(* CODESYS project e!C_BasicProg_1.ECP

Project tree, tasks and I/O mapping:
  PFC8203 : 750-8203 PFC200 2ETH CAN, WAGO, order no. 0750-8203, version 5.11.1.16
    application Application
      libraries: Standard, * (System); Util, * (System)
      task Test (cyclic, interval T#10ms, priority 11) calls PLC_PRG
      task VISU_TASK (cyclic, interval 100 ms, priority 15) calls VisuElems.Visu_Prg
      Data types/
        data type typControlInterface
      Global Variables/
        global variables Variable_Configuration
        global variables GVL
      POUs/
        CASE_OF/
          program Template_CASE_OF [ST]
          program Test1_CASE_OF [ST]
        FB_POINTER/
          function block fbPointerControl [ST]
          program Template_FB_POINTER [ST]
          program Test1_FB_POINTER [ST]
        FB_STRUCT/
          function block fbStructControl [ST]
          program Template_FB_STRUCT [ST]
          program Test1_FB_STRUCT [ST]
        FOR_DO_ARRAY/
          program Template_FOR_DO_ARRAY [ST]: Action1_ST, Action2_ST, Action3_ST
          program Test1_FOR_DO_ARRAY [ST]: Action1_ST, Action2_ST, Action3_ST
        program PLC_PRG [ST]
        IF_THEN_ELSE/
          program Test1_IF_THEN_ELSE [ST]: Action3_CFC, Action1_ST, Action2_SFC, ActivationMonitoring_active, Inactivation_active, Init_active, OutputControl_active
          program Template_IF_THEN_ELSE [ST]: Action2_SFC, Action3_CFC, Action1_ST, Inactivation_active, ActivationMonitoring_active, OutputControl_active, Init_active
      Visualizations/
        visualisation FB_STRUCT
        visualisation IF_THEN_ELSE
      global variables PersistentVars
      trace Sampling_Trace (task Test): Test_FB_STRUCT.typEngineControl.rControlPosition, Test1_FOR_DO_ARRAY.rSineSample
    DeviceAdapter
    Kbus : Kbus, WAGO, version 1.4.0.2
        unmapped channels: K-BUS diagnostics
    MODBUS
      MODBUS : MODBUS, WAGO, order no. n/a, version 1.1.1.15
    CANbus
  libraries: Util, 3.5.11.0 (System); VisuSymbols, 3.5.10.0 (System); WagoVisuIcons, 1.0.0.8 (WAGO)
  GlobalImagePool
  text list GlobalTextList
*)

// PFC8203/Application/Data types/typControlInterface
TYPE typControlInterface :
STRUCT
	TON_ControlDelay: TON;
	R_TRIG_ControlStart: R_TRIG;
	R_TRIG_ControlStop: R_TRIG;
	tControlDelay: TIME := T#2s;
	xControlEnable: BOOL;
	xControlRun: BOOL;
	xControlStart: BOOL;
	xControlStop: BOOL;
	xControlOut: BOOL;

	GEN_ControlSimulator: GEN;
	SimulatorMode: GEN_MODE;
	SimulatorPeriod: TIME := T#2s;
	SimulatorAmplitude: INT := 100;
	rSimulatorLimit: REAL := 100.0;
	rSimulatorLevel: REAL := 100.1;
	rSimulatorPosition: REAL;
END_STRUCT
END_TYPE

// PFC8203/Application/Global Variables/Variable_Configuration
VAR_CONFIG
END_VAR

// PFC8203/Application/PersistentVars
VAR_GLOBAL PERSISTENT RETAIN
END_VAR

// PFC8203/Application/Global Variables/GVL
VAR_GLOBAL
END_VAR

// PFC8203/Application/POUs/PLC_PRG
PROGRAM PLC_PRG
VAR
END_VAR



Template_IF_THEN_ELSE();
Test1_IF_THEN_ELSE();

Template_CASE_OF();
Test1_CASE_OF();


Template_FOR_DO_ARRAY();
Test1_FOR_DO_ARRAY();


Template_FB_STRUCT();
Test1_FB_STRUCT();


Template_FB_POINTER();
Test1_FB_POINTER();

END_PROGRAM

// PFC8203/Application/POUs/IF_THEN_ELSE/Template_IF_THEN_ELSE
PROGRAM Template_IF_THEN_ELSE
VAR
	TON_ControlDelay_1: TON;
	R_TRIG_ControlStart_1: R_TRIG;
	R_TRIG_ControlStop_1: R_TRIG;
	tControlDelay_1: TIME := T#2s;
	xControlEnable_1: BOOL;
	xControlRun_1: BOOL;
	xControlStart_1: BOOL;
	xControlStop_1: BOOL;
	xControlOut_1: BOOL;

	TON_ControlDelay_2: TON;
	R_TRIG_ControlStart_2: R_TRIG;
	R_TRIG_ControlStop_2: R_TRIG;
	tControlDelay_2: TIME := T#2s;
	xControlEnable_2: BOOL;
	xControlRun_2: BOOL;
	xControlStart_2: BOOL;
	xControlStop_2: BOOL;
	xControlOut_2: BOOL;

	TON_ControlDelay_3: TON;
	R_TRIG_ControlStart_3: R_TRIG;
	R_TRIG_ControlStop_3: R_TRIG;
	tControlDelay_3: TIME := T#2s;
	xControlEnable_3: BOOL;
	xControlRun_3: BOOL;
	xControlStart_3: BOOL;
	xControlStop_3: BOOL;
	xControlOut_3: BOOL;

END_VAR
VAR // added by the converter: edge detectors and wires of the graphical bodies
    _w1 : BOOL;
END_VAR



Action1_ST();

Action2_SFC();

Action3_CFC();

ACTION Action2_SFC:
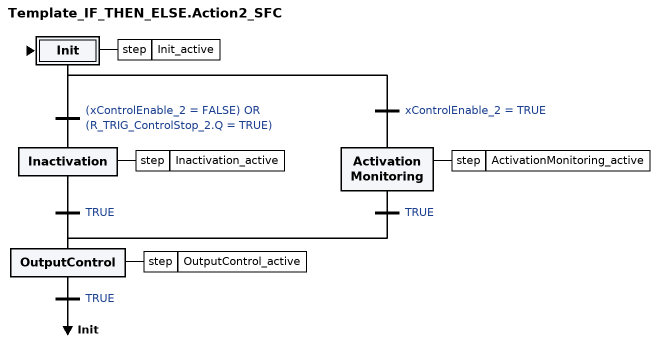
INITIAL_STEP Init:
    Init_active(N);  // step action
END_STEP
TRANSITION FROM Init TO Inactivation
    := (xControlEnable_2 = FALSE) OR (R_TRIG_ControlStop_2.Q = TRUE);
END_TRANSITION
STEP Inactivation:
    Inactivation_active(N);  // step action
END_STEP
TRANSITION FROM Inactivation TO OutputControl
    := TRUE;
END_TRANSITION
TRANSITION FROM Init TO ActivationMonitoring
    := xControlEnable_2 = TRUE;
END_TRANSITION
STEP ActivationMonitoring:
    ActivationMonitoring_active(N);  // step action
END_STEP
TRANSITION FROM ActivationMonitoring TO OutputControl
    := TRUE;
END_TRANSITION
STEP OutputControl:
    OutputControl_active(N);  // step action
END_STEP
TRANSITION FROM OutputControl TO Init
    := TRUE;
END_TRANSITION
// branch label Branch1_Action2_SFC
END_ACTION

ACTION Action3_CFC:
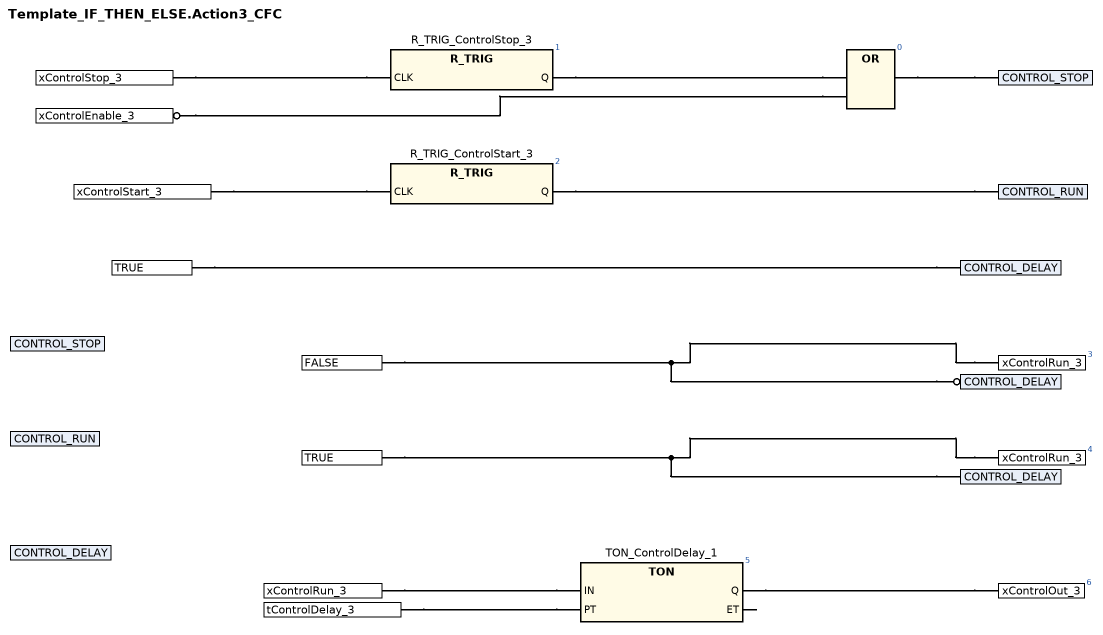
(* R_TRIG_ControlStop_3.Q OR NOT xControlEnable_3; result not used *)
R_TRIG_ControlStop_3(CLK := xControlStop_3); // R_TRIG
R_TRIG_ControlStart_3(CLK := xControlStart_3); // R_TRIG
xControlRun_3 := FALSE;
xControlRun_3 := TRUE;
TON_ControlDelay_1(IN := xControlRun_3, PT := tControlDelay_3); // TON
xControlOut_3 := TON_ControlDelay_1.Q;
END_ACTION

ACTION Action1_ST:


(* Monitor start/stop signal for output activation/inactivation *)
R_TRIG_ControlStart_1(CLK:= xControlStart_1);
R_TRIG_ControlStop_1(CLK:= xControlStop_1);
IF ((xControlEnable_1 = FALSE) OR (R_TRIG_ControlStop_1.Q = TRUE))THEN
	xControlRun_1 := FALSE;
ELSE
	IF (R_TRIG_ControlStart_1.Q = TRUE) THEN
		xControlRun_1 := TRUE;
	END_IF
END_IF


(* Activate output after specified delay *)
TON_ControlDelay_1(IN:= xControlRun_1, PT:= tControlDelay_1, Q=> xControlOut_1);
END_ACTION

ACTION Inactivation_active:
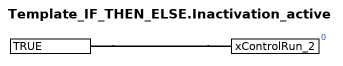
xControlRun_2 := TRUE;
END_ACTION

ACTION ActivationMonitoring_active:
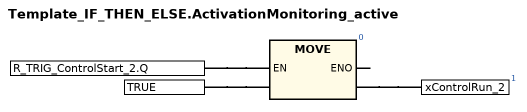
IF R_TRIG_ControlStart_2.Q THEN _w1 := TRUE; END_IF
xControlRun_2 := _w1;
END_ACTION

ACTION OutputControl_active:
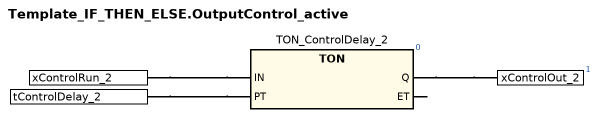
TON_ControlDelay_2(IN := xControlRun_2, PT := tControlDelay_2); // TON
xControlOut_2 := TON_ControlDelay_2.Q;
END_ACTION

ACTION Init_active:
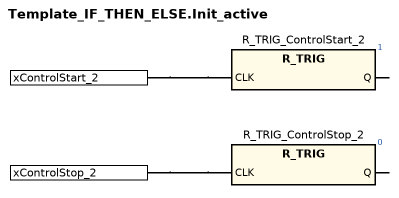
R_TRIG_ControlStop_2(CLK := xControlStop_2); // R_TRIG
R_TRIG_ControlStart_2(CLK := xControlStart_2); // R_TRIG
END_ACTION

END_PROGRAM

// PFC8203/Application/POUs/IF_THEN_ELSE/Test1_IF_THEN_ELSE
PROGRAM Test1_IF_THEN_ELSE
VAR
	TON_ControlDelay_1: TON;
	R_TRIG_ControlStart_1: R_TRIG;
	R_TRIG_ControlStop_1: R_TRIG;
	tControlDelay_1: TIME := T#2s;
	xControlEnable_1: BOOL;
	xControlRun_1: BOOL;
	xControlStart_1: BOOL;
	xControlStop_1: BOOL;
	xControlOut_1: BOOL;

	TON_ControlDelay_2: TON;
	R_TRIG_ControlStart_2: R_TRIG;
	R_TRIG_ControlStop_2: R_TRIG;
	tControlDelay_2: TIME := T#2s;
	xControlEnable_2: BOOL;
	xControlRun_2: BOOL;
	xControlStart_2: BOOL;
	xControlStop_2: BOOL;
	xControlOut_2: BOOL;

	TON_ControlDelay_3: TON;
	R_TRIG_ControlStart_3: R_TRIG;
	R_TRIG_ControlStop_3: R_TRIG;
	tControlDelay_3: TIME := T#2s;
	xControlEnable_3: BOOL;
	xControlRun_3: BOOL;
	xControlStart_3: BOOL;
	xControlStop_3: BOOL;
	xControlOut_3: BOOL;

END_VAR
VAR // added by the converter: edge detectors and wires of the graphical bodies
    _w1 : BOOL;
END_VAR



Action1_ST();

Action2_SFC();

Action3_CFC();

ACTION Action3_CFC:
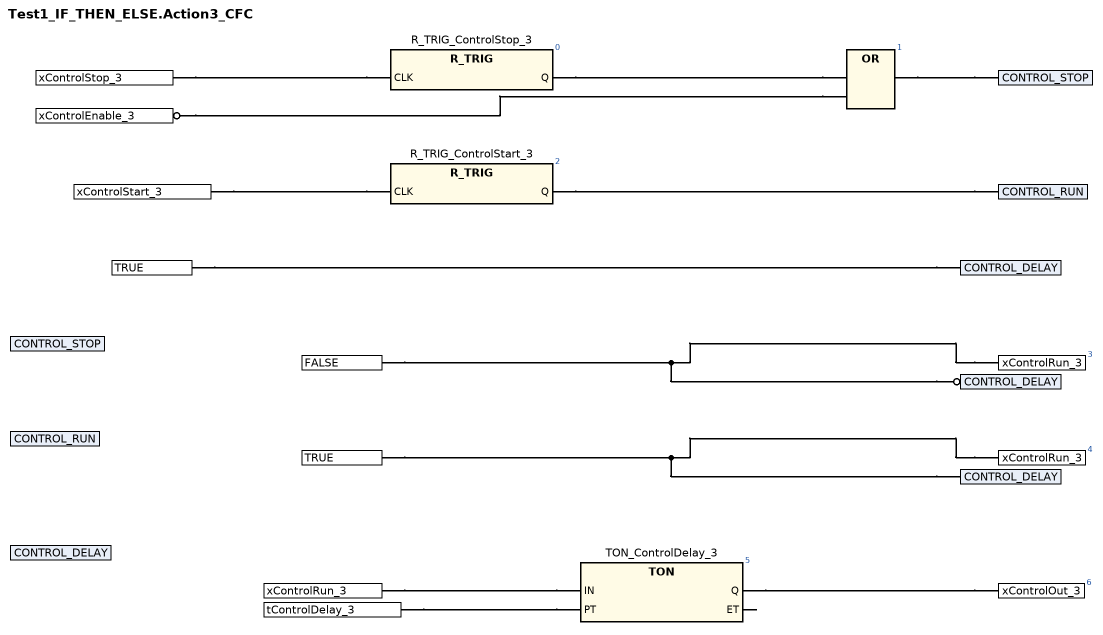
R_TRIG_ControlStop_3(CLK := xControlStop_3); // R_TRIG
(* R_TRIG_ControlStop_3.Q OR NOT xControlEnable_3; result not used *)
R_TRIG_ControlStart_3(CLK := xControlStart_3); // R_TRIG
xControlRun_3 := FALSE;
xControlRun_3 := TRUE;
TON_ControlDelay_3(IN := xControlRun_3, PT := tControlDelay_3); // TON
xControlOut_3 := TON_ControlDelay_3.Q;
END_ACTION

ACTION Action1_ST:


(* Monitor start/stop signal for output activation/inactivation *)
R_TRIG_ControlStart_1(CLK:= xControlStart_1);
R_TRIG_ControlStop_1(CLK:= xControlStop_1);
IF ((xControlEnable_1 = FALSE) OR (R_TRIG_ControlStop_1.Q = TRUE))THEN
	xControlRun_1 := FALSE;
ELSE
	IF (R_TRIG_ControlStart_1.Q = TRUE) THEN
		xControlRun_1 := TRUE;
	END_IF
END_IF


(* Activate output after specified delay *)
TON_ControlDelay_1(IN:= xControlRun_1, PT:= tControlDelay_1, Q=> xControlOut_1);
END_ACTION

ACTION Action2_SFC:
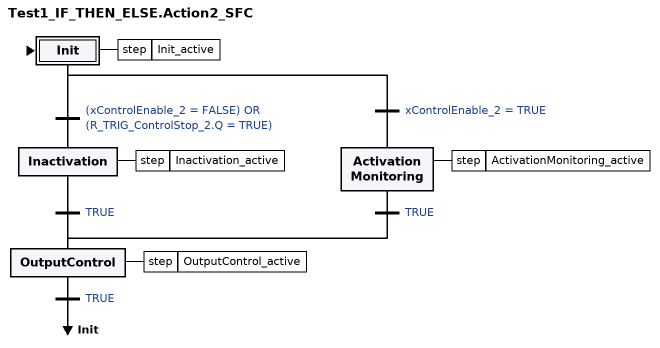
INITIAL_STEP Init:
    Init_active(N);  // step action
END_STEP
TRANSITION FROM Init TO Inactivation
    := (xControlEnable_2 = FALSE) OR (R_TRIG_ControlStop_2.Q = TRUE);
END_TRANSITION
STEP Inactivation:
    Inactivation_active(N);  // step action
END_STEP
TRANSITION FROM Inactivation TO OutputControl
    := TRUE;
END_TRANSITION
TRANSITION FROM Init TO ActivationMonitoring
    := xControlEnable_2 = TRUE;
END_TRANSITION
STEP ActivationMonitoring:
    ActivationMonitoring_active(N);  // step action
END_STEP
TRANSITION FROM ActivationMonitoring TO OutputControl
    := TRUE;
END_TRANSITION
STEP OutputControl:
    OutputControl_active(N);  // step action
END_STEP
TRANSITION FROM OutputControl TO Init
    := TRUE;
END_TRANSITION
// branch label Branch1_Action2_SFC
END_ACTION

ACTION ActivationMonitoring_active:
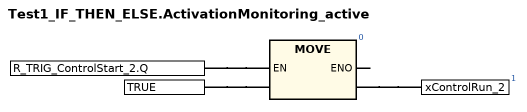
IF R_TRIG_ControlStart_2.Q THEN _w1 := TRUE; END_IF
xControlRun_2 := _w1;
END_ACTION

ACTION Inactivation_active:
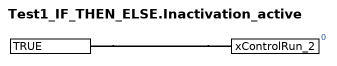
xControlRun_2 := TRUE;
END_ACTION

ACTION Init_active:
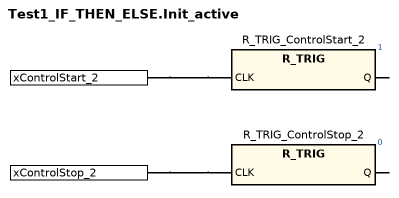
R_TRIG_ControlStop_2(CLK := xControlStop_2); // R_TRIG
R_TRIG_ControlStart_2(CLK := xControlStart_2); // R_TRIG
END_ACTION

ACTION OutputControl_active:
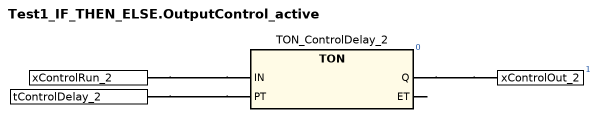
TON_ControlDelay_2(IN := xControlRun_2, PT := tControlDelay_2); // TON
xControlOut_2 := TON_ControlDelay_2.Q;
END_ACTION

END_PROGRAM

// PFC8203/Application/POUs/CASE_OF/Template_CASE_OF
PROGRAM Template_CASE_OF
VAR
	TON_ControlDelay: TON;
	R_TRIG_ControlStart: R_TRIG;
	R_TRIG_ControlStop: R_TRIG;
	tControlDelay: TIME := T#2s;
	wControlState: WORD;
	xControlEnable: BOOL;
	xControlRun: BOOL;
	xControlStart: BOOL;
	xControlStop: BOOL;
	xControlOut: BOOL;
END_VAR



R_TRIG_ControlStart(CLK:= xControlStart);
R_TRIG_ControlStop(CLK:= xControlStop);

(* Monitor signal activation sequence *)
CASE wControlState OF

	0:(* Init signal monitoring *)
		wControlState := 10;

	10:(* Signal currently active, wait for inactivation *)
		IF ((xControlEnable = FALSE) OR (R_TRIG_ControlStop.Q = TRUE)) THEN
			xControlRun := FALSE;
			wControlState := 20;
		END_IF

	20:(* Signal currently incative, wait for activation *)
		IF ((xControlEnable = TRUE) AND (R_TRIG_ControlStart.Q = TRUE)) THEN
			xControlRun := TRUE;
			wControlState := 10;
		END_IF

END_CASE


(* Activate output after specified delay when commanded *)
TON_ControlDelay(IN:= xControlRun, PT:= tControlDelay, Q=> xControlOut);

END_PROGRAM

// PFC8203/Application/POUs/CASE_OF/Test1_CASE_OF
PROGRAM Test1_CASE_OF
VAR
	TON_ControlDelay: TON;
	R_TRIG_ControlStart: R_TRIG;
	R_TRIG_ControlStop: R_TRIG;
	tControlDelay: TIME := T#2s;
	wControlState: WORD;
	xControlEnable: BOOL;
	xControlRun: BOOL;
	xControlStart: BOOL;
	xControlStop: BOOL;
	xControlOut: BOOL;
END_VAR



R_TRIG_ControlStart(CLK:= xControlStart);
R_TRIG_ControlStop(CLK:= xControlStop);

(* Monitor signal activation sequence *)
CASE wControlState OF

	0:(* Init signal monitoring *)
		wControlState := 10;

	10:(* Signal currently active, wait for inactivation *)
		IF ((xControlEnable = FALSE) OR (R_TRIG_ControlStop.Q = TRUE)) THEN
			xControlRun := FALSE;
			wControlState := 20;
		END_IF

	20:(* Signal currently incative, wait for activation *)
		IF ((xControlEnable = TRUE) AND (R_TRIG_ControlStart.Q = TRUE)) THEN
			xControlRun := TRUE;
			wControlState := 10;
		END_IF

END_CASE


(* Activate output after specified delay when commanded *)
TON_ControlDelay(IN:= xControlRun, PT:= tControlDelay, Q=> xControlOut);

END_PROGRAM

// PFC8203/Application/POUs/FOR_DO_ARRAY/Template_FOR_DO_ARRAY
PROGRAM Template_FOR_DO_ARRAY
VAR CONSTANT
	iArrayLimit1: INT := 9;
	iArrayLimit2: INT := 9;
	iArrayLimit3: INT := 19;
	iArrayLimit4: INT := 49;
	iModuloLimit: INT := 50;
END_VAR
VAR
	iArrayIndex: INT;
	dwCnt: DWORD;
	wCnt: WORD;
	awArrayTest1: ARRAY[0..iArrayLimit1] OF WORD;
	adwArrayTest2 AT %MW0 : ARRAY[0..iArrayLimit2] OF DWORD;
	awArrayTest3 AT %MW0 : ARRAY[0..iArrayLimit3] OF WORD;

	iArrayIndexModulo: INT;
	TON_SineSampler: TON;
	tSineInterval: TIME := T#200ms;
	rSineAngle: REAL;
	rSineSample: REAL;
	arSineArray: ARRAY[0..iArrayLimit4] OF REAL;

	TON_ControlDelay: ARRAY[0..iArrayLimit1] OF TON;
	R_TRIG_ControlStart: ARRAY[0..iArrayLimit1] OF R_TRIG;
	R_TRIG_ControlStop: ARRAY[0..iArrayLimit1] OF R_TRIG;
	tControlDelay: ARRAY[0..iArrayLimit1] OF TIME := [iArrayLimit1(T#2S)];
	xControlEnable: ARRAY[0..iArrayLimit1] OF BOOL;
	xControlRun: ARRAY[0..iArrayLimit1] OF BOOL;
	xControlStart: ARRAY[0..iArrayLimit1] OF BOOL;
	xControlStop: ARRAY[0..iArrayLimit1] OF BOOL;
	xControlOut: ARRAY[0..iArrayLimit1] OF BOOL;
END_VAR


Action1_ST();

Action2_ST();

Action3_ST();

ACTION Action1_ST:

(* Run same logic for all array elements *)
FOR iArrayIndex := 0 TO iArrayLimit1 DO

	wCnt := wCnt + 1;
	dwCnt := dwCnt + 1;

	awArrayTest1[iArrayIndex] := wCnt;

	adwArrayTest2[iArrayIndex] := dwCnt;

	awArrayTest3[2*iArrayIndex] := DWORD_TO_WORD(dwCnt);
	awArrayTest3[(2*iArrayIndex)+1] := DWORD_TO_WORD(SHR(dwCnt, 16));

END_FOR
END_ACTION

ACTION Action2_ST:

(* Run same logic for all array elements *)
FOR iArrayIndex := 0 TO iArrayLimit1 DO

	(* Monitor start/stop signal for output activation/inactivation *)
	R_TRIG_ControlStart[iArrayIndex](CLK:= xControlStart[iArrayIndex]);
	R_TRIG_ControlStop[iArrayIndex](CLK:= xControlStop[iArrayIndex]);
	IF ((xControlEnable[iArrayIndex] = FALSE) OR (R_TRIG_ControlStop[iArrayIndex].Q = TRUE))THEN
		xControlRun[iArrayIndex] := FALSE;
	ELSE
		IF (R_TRIG_ControlStart[iArrayIndex].Q = TRUE) THEN
			xControlRun[iArrayIndex] := TRUE;
		END_IF
	END_IF
	
	(* Activate output after specified delay *)
	TON_ControlDelay[iArrayIndex](IN:= xControlRun[iArrayIndex], PT:= tControlDelay[iArrayIndex], Q=> xControlOut[iArrayIndex]);

END_FOR
END_ACTION

ACTION Action3_ST:

rSineAngle := DWORD_TO_REAL(REAL_TO_DWORD((rSineAngle + 0.1)*100) MOD REAL_TO_DWORD(2*3.14159265358*100));
rSineSample := SIN(rSineAngle);
TON_SineSampler(IN:= TRUE, PT:= tSineInterval);
IF(TON_SineSampler.Q = TRUE) THEN
	TON_SineSampler(IN:= FALSE);
	arSineArray[iArrayIndexModulo] := rSineSample;
	iArrayIndexModulo := (iArrayIndexModulo + 1) MOD iModuloLimit;
END_IF
END_ACTION

END_PROGRAM

// PFC8203/Application/POUs/FOR_DO_ARRAY/Test1_FOR_DO_ARRAY
PROGRAM Test1_FOR_DO_ARRAY
VAR CONSTANT
	iArrayLimit1: INT := 9;
	iArrayLimit2: INT := 9;
	iArrayLimit3: INT := 19;
	iArrayLimit4: INT := 49;
	iModuloLimit: INT := 50;
END_VAR
VAR
	iArrayIndex: INT;
	dwCnt: DWORD;
	wCnt: WORD;
	awArrayTest1: ARRAY[0..iArrayLimit1] OF WORD;
	adwArrayTest2 AT %MW0 : ARRAY[0..iArrayLimit2] OF DWORD;
	awArrayTest3 AT %MW0 : ARRAY[0..iArrayLimit3] OF WORD;

	iArrayIndexModulo: INT;
	TON_SineSampler: TON;
	tSineInterval: TIME := T#200ms;
	rSineAngle: REAL;
	rSineSample: REAL;
	arSineArray: ARRAY[0..iArrayLimit4] OF REAL;

	TON_ControlDelay: ARRAY[0..iArrayLimit1] OF TON;
	R_TRIG_ControlStart: ARRAY[0..iArrayLimit1] OF R_TRIG;
	R_TRIG_ControlStop: ARRAY[0..iArrayLimit1] OF R_TRIG;
	tControlDelay: ARRAY[0..iArrayLimit1] OF TIME := [iArrayLimit1(T#2S)];
	xControlEnable: ARRAY[0..iArrayLimit1] OF BOOL;
	xControlRun: ARRAY[0..iArrayLimit1] OF BOOL;
	xControlStart: ARRAY[0..iArrayLimit1] OF BOOL;
	xControlStop: ARRAY[0..iArrayLimit1] OF BOOL;
	xControlOut: ARRAY[0..iArrayLimit1] OF BOOL;
END_VAR


Action1_ST();

Action2_ST();

Action3_ST();

ACTION Action1_ST:

(* Run same logic for all array elements *)
FOR iArrayIndex := 0 TO iArrayLimit1 DO

	wCnt := wCnt + 1;
	dwCnt := dwCnt + 1;

	awArrayTest1[iArrayIndex] := wCnt;

	adwArrayTest2[iArrayIndex] := dwCnt;

	awArrayTest3[2*iArrayIndex] := DWORD_TO_WORD(dwCnt);
	awArrayTest3[(2*iArrayIndex)+1] := DWORD_TO_WORD(SHR(dwCnt, 16));

END_FOR
END_ACTION

ACTION Action2_ST:

(* Run same logic for all array elements *)
FOR iArrayIndex := 0 TO iArrayLimit1 DO

	(* Monitor start/stop signal for output activation/inactivation *)
	R_TRIG_ControlStart[iArrayIndex](CLK:= xControlStart[iArrayIndex]);
	R_TRIG_ControlStop[iArrayIndex](CLK:= xControlStop[iArrayIndex]);
	IF ((xControlEnable[iArrayIndex] = FALSE) OR (R_TRIG_ControlStop[iArrayIndex].Q = TRUE))THEN
		xControlRun[iArrayIndex] := FALSE;
	ELSE
		IF (R_TRIG_ControlStart[iArrayIndex].Q = TRUE) THEN
			xControlRun[iArrayIndex] := TRUE;
		END_IF
	END_IF
	
	(* Activate output after specified delay *)
	TON_ControlDelay[iArrayIndex](IN:= xControlRun[iArrayIndex], PT:= tControlDelay[iArrayIndex], Q=> xControlOut[iArrayIndex]);

END_FOR
END_ACTION

ACTION Action3_ST:

rSineAngle := DWORD_TO_REAL(REAL_TO_DWORD((rSineAngle + 0.1)*100) MOD REAL_TO_DWORD(2*3.14159265358*100));
rSineSample := SIN(rSineAngle);
TON_SineSampler(IN:= TRUE, PT:= tSineInterval);
IF(TON_SineSampler.Q = TRUE) THEN
	TON_SineSampler(IN:= FALSE);
	arSineArray[iArrayIndexModulo] := rSineSample;
	iArrayIndexModulo := (iArrayIndexModulo + 1) MOD iModuloLimit;
END_IF
END_ACTION

END_PROGRAM

// PFC8203/Application/POUs/FB_STRUCT/Template_FB_STRUCT
PROGRAM Template_FB_STRUCT
VAR CONSTANT
	LIM_OF_VALVES : INT := 9;
END_VAR
VAR
	fbEngineControl: fbStructControl;
	typEngineControl: typControlInterface;

	fbEnginePump: fbStructControl;
	typPumpControl: typControlInterface;

	afbValveControl: ARRAY[0..LIM_OF_VALVES] OF fbStructControl;
	atypValveControl: ARRAY[0..LIM_OF_VALVES] OF typControlInterface;
	iValveIndex: INT;

	typVisuControl: typControlInterface;
	iVisuValveIndex: INT;
END_VAR


(* Initialize struct elements *)
(*typEngineControl.xControlEnable := TRUE;
typEngineControl.xControlStart := TRUE;*)
typEngineControl.tControlDelay := T#2s;
typEngineControl.rSimulatorLimit := 100.0;
typEngineControl.rSimulatorLevel := 100.1;

(* Run struct action  *)
fbEnginePump(typControlInterface:= typPumpControl);


(* Initialize struct elements *)
(*typPumpControl.xControlEnable := TRUE;
typPumpControl.xControlStart := TRUE;*)
typPumpControl.tControlDelay := T#5s;
typPumpControl.rSimulatorLimit := 100.0;
typPumpControl.rSimulatorLevel := 100.1;

(* Run struct action  *)
fbEngineControl(typControlInterface:= typEngineControl);


(* Run same action for all structs in the array *)
FOR iValveIndex := 0 TO LIM_OF_VALVES DO
	(*
	IF (iValveIndex < 6) THEN
		atypValveControl[iValveIndex].xControlEnable := TRUE;
	END_IF
	*)
	atypValveControl[iValveIndex].tControlDelay := T#2s;
	atypValveControl[iValveIndex].rSimulatorLimit := 100.0;
	atypValveControl[iValveIndex].rSimulatorLevel := 100.1;
	afbValveControl[iValveIndex](typControlInterface:= atypValveControl[iValveIndex]);
END_FOR


(* For visu only *)
atypValveControl[iVisuValveIndex].xControlEnable := typVisuControl.xControlEnable;
atypValveControl[iVisuValveIndex].xControlStart := typVisuControl.xControlStart;
atypValveControl[iVisuValveIndex].xControlStop := typVisuControl.xControlStop;
typVisuControl.xControlOut := atypValveControl[iVisuValveIndex].xControlOut;
typVisuControl.TON_ControlDelay := atypValveControl[iVisuValveIndex].TON_ControlDelay;

END_PROGRAM

// PFC8203/Application/POUs/FB_STRUCT/fbStructControl
FUNCTION_BLOCK fbStructControl
VAR_IN_OUT
	typControlInterface: typControlInterface;
END_VAR



(* Monitor start/stop signal for output activation/inactivation *)
typControlInterface.R_TRIG_ControlStart(CLK:= typControlInterface.xControlStart);
typControlInterface.R_TRIG_ControlStop(CLK:= typControlInterface.xControlStop);
IF ((typControlInterface.xControlEnable = FALSE) OR (typControlInterface.R_TRIG_ControlStop.Q = TRUE))THEN
	typControlInterface.xControlRun := FALSE;
ELSE
	IF (typControlInterface.R_TRIG_ControlStart.Q = TRUE) THEN
		typControlInterface.xControlRun := TRUE;
	END_IF
END_IF

(* Activate output after specified delay *)
typControlInterface.TON_ControlDelay(IN:= typControlInterface.xControlRun, PT:= typControlInterface.tControlDelay, Q=> typControlInterface.xControlOut);



(* Run simulator functionality *)
IF (typControlInterface.xControlEnable = TRUE) THEN
	typControlInterface.GEN_ControlSimulator(
		MODE		:= typControlInterface.SimulatorMode,
		BASE		:= TRUE,
		PERIOD		:= typControlInterface.SimulatorPeriod,
		CYCLES		:= ,
		AMPLITUDE	:= typControlInterface.SimulatorAmplitude,
		RESET		:= ,
		OUT			=> );
END_IF
typControlInterface.rSimulatorPosition := INT_TO_REAL(100 + typControlInterface.GEN_ControlSimulator.OUT);

END_FUNCTION_BLOCK

// PFC8203/Application/POUs/FB_STRUCT/Test1_FB_STRUCT
PROGRAM Test1_FB_STRUCT
VAR CONSTANT
	LIM_OF_VALVES : INT := 9;
END_VAR
VAR
	fbEngineControl: fbStructControl;
	typEngineControl: typControlInterface;

	fbEnginePump: fbStructControl;
	typPumpControl: typControlInterface;

	afbValveControl: ARRAY[0..LIM_OF_VALVES] OF fbStructControl;
	atypValveControl: ARRAY[0..LIM_OF_VALVES] OF typControlInterface;
	iValveIndex: INT;

END_VAR


(* Initialize struct elements *)
(*typEngineControl.xControlEnable := TRUE;
typEngineControl.xControlStart := TRUE;*)
typEngineControl.tControlDelay := T#2s;
typEngineControl.rSimulatorLimit := 100.0;
typEngineControl.rSimulatorLevel := 100.1;

(* Run struct action  *)
fbEnginePump(typControlInterface:= typPumpControl);


(* Initialize struct elements *)
(*typPumpControl.xControlEnable := TRUE;
typPumpControl.xControlStart := TRUE;*)
typPumpControl.tControlDelay := T#5s;
typPumpControl.rSimulatorLimit := 100.0;
typPumpControl.rSimulatorLevel := 100.1;

(* Run struct action  *)
fbEngineControl(typControlInterface:= typEngineControl);


(* Run same action for all structs in the array *)
FOR iValveIndex := 0 TO LIM_OF_VALVES DO
	IF (iValveIndex < 6) THEN
		atypValveControl[iValveIndex].xControlEnable := TRUE;
	END_IF
	atypValveControl[iValveIndex].tControlDelay := T#2s;
	atypValveControl[iValveIndex].rSimulatorLimit := 100.0;
	atypValveControl[iValveIndex].rSimulatorLevel := 100.1;
	afbValveControl[iValveIndex](typControlInterface:= atypValveControl[iValveIndex]);
END_FOR

END_PROGRAM

// PFC8203/Application/POUs/FB_POINTER/Template_FB_POINTER
PROGRAM Template_FB_POINTER
VAR CONSTANT
	iArrayLimit: INT := 9;
END_VAR
VAR
	awArrayTest: ARRAY[0..iArrayLimit] OF WORD;
	fbControlInit : fbPointerControl;
END_VAR



(* Run same logic for all array elements *)
fbControlInit(pawArrayTest:= ADR(awArrayTest[0]), iArrayLimit:= iArrayLimit);

END_PROGRAM

// PFC8203/Application/POUs/FB_POINTER/fbPointerControl
FUNCTION_BLOCK fbPointerControl
VAR_INPUT
	pawArrayTest: POINTER TO ARRAY[0..1000(* dummy size *)] OF WORD;
	iArrayLimit: INT := 0;
END_VAR
VAR
	iArrayIndex: INT;
	pwArrayTest: POINTER TO WORD;
	pwArrayIndex: POINTER TO WORD;
END_VAR


(* Run same logic for all array elements, array size not pre-defined *)
pwArrayIndex := 0;
FOR iArrayIndex := 0 TO iArrayLimit DO

	(* Alternative 1: *)
	pawArrayTest^[iArrayIndex] := iArrayIndex*10;

	(* Alternative 2: *)
	pwArrayTest := pawArrayTest+pwArrayIndex;
	pwArrayTest^ := iArrayIndex;
	pwArrayIndex := pwArrayIndex+2;

END_FOR

END_FUNCTION_BLOCK

// PFC8203/Application/POUs/FB_POINTER/Test1_FB_POINTER
PROGRAM Test1_FB_POINTER
VAR CONSTANT
	iArrayLimit: INT := 9;
END_VAR
VAR
	awArrayTest: ARRAY[0..iArrayLimit] OF WORD;
	fbControlInit : fbPointerControl;
END_VAR



(* Run same logic for all array elements *)
fbControlInit(pawArrayTest:= ADR(awArrayTest[0]), iArrayLimit:= iArrayLimit);

END_PROGRAM

// PFC8203/Application/Visualizations/FB_STRUCT
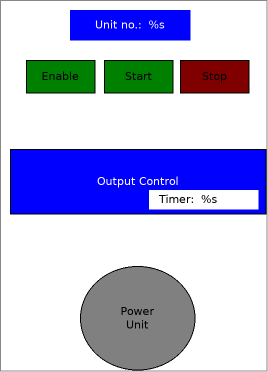
VISUALIZATION FB_STRUCT  // 268x372
    RoundedRectangle (10,149 256x65), "Output Control"
    Ellipse (80,266 115x104), "Power Unit", colour toggle: Template_FB_STRUCT.typVisuControl.xControlOut
    RoundedRectangle (104,60 69x33), "Start", colour toggle: Template_FB_STRUCT.typVisuControl.xControlStart
        tap Template_FB_STRUCT.typVisuControl.xControlStart
    RoundedRectangle (180,60 69x33), "Stop", colour toggle: Template_FB_STRUCT.typVisuControl.xControlStop
        tap Template_FB_STRUCT.typVisuControl.xControlStop
    RoundedRectangle (26,60 69x33), "Enable", colour toggle: Template_FB_STRUCT.typVisuControl.xControlEnable
        toggle Template_FB_STRUCT.typVisuControl.xControlEnable
    RoundedRectangle (149,190 109x19), "Timer: %s", text variable: Template_FB_STRUCT.typVisuControl.TON_ControlDelay.ET
    Polygon (57,137)
    Polygon (133,137)
    Polygon (211,137)
    Polygon (133,257)
    RoundedRectangle (70,10 120x30), "Unit no.: %s", text variable: Template_FB_STRUCT.iVisuValveIndex
        OnMouseDown: write the text variable via Edit, min 0, max 9
END_VISUALIZATION

// PFC8203/Application/Visualizations/IF_THEN_ELSE
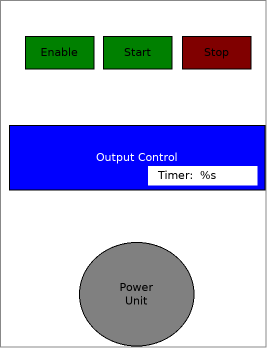
VISUALIZATION IF_THEN_ELSE  // 267x348
    RoundedRectangle (9,125 256x65), "Output Control"
    Ellipse (79,242 115x104), "Power Unit", colour toggle: (Template_IF_THEN_ELSE.xControlOut_1) <> 0
    RoundedRectangle (103,36 69x33), "Start", colour toggle: (Template_IF_THEN_ELSE.xControlStart_1) <> 0
        tap Template_IF_THEN_ELSE.xControlStart_1
    RoundedRectangle (182,36 69x33), "Stop", colour toggle: (Template_IF_THEN_ELSE.xControlStop_1) <> 0
        tap Template_IF_THEN_ELSE.xControlStop_1
    RoundedRectangle (25,36 69x33), "Enable", colour toggle: (Template_IF_THEN_ELSE.xControlEnable_1) <> 0
        toggle Template_IF_THEN_ELSE.xControlEnable_1
    RoundedRectangle (148,166 109x19), "Timer: %s", text variable: Template_IF_THEN_ELSE.TON_ControlDelay_1.ET
    Polygon (56,113)
    Polygon (132,113)
    Polygon (210,113)
    Polygon (132,233)
END_VISUALIZATION
